// TIA Portal project "ANALOG INPUT" (V19)

(* hardware
DEVICE "SIMATIC 1200 station_1"  S71200.Device
   slot 0: "S7-1200 rack"  Rack  V1.0
   slot 1: "PLC_1"  CPU 1214C DC/DC/DC  6ES7 214-1AG40-0XB0  V4.0
   slot 3: "AQ1 x 12 bits_1"  6ES7 232-4HA30-0XB0  V1.0
DEVICE "HMI_1"  KTP600 Basic color PN
   slot 0: "HMI"  HMI  6AV6 647-0AD11-3AX0  12.0.0.0
   slot 1: "HMI_RT_1"  KTP600 Basic color PN  6AV6 647-0AD11-3AX0  12.0.0.0
   slot 5: "IE_CP_1"  PROFINET Interface  IE_CP  V7.1.0
      slot 1: "PROFINET_Interface_1"  PROFINET Interface
         slot 1: "PORT_1"  Port  1.0.0.0
*)

// ===== PLC "PLC_1"  CPU 1214C DC/DC/DC =====

DATA_BLOCK "Simulated Analog Input"   // DB1
{ S7_Optimized_Access := 'TRUE' }
VERSION : 0.1
   VAR
      HEIGHT_AI : Int;
   END_VAR
BEGIN
END_DATA_BLOCK

ORGANIZATION_BLOCK "Main"   // OB1, LAD, ProgramCycle
TITLE = "Main Program Sweep (Cycle)"
{ S7_Optimized_Access := 'TRUE' }
VERSION : 0.1
BEGIN
END_ORGANIZATION_BLOCK

(* ===== HMI "HMI_RT_1" =====
system functions are stored by id; their names below are inferred from use
connection "HMI_Connection_1": ETHERNET, SMART_S7_1200_OMS

HMI tags "Default tag table"
   "Conveyor_Control_DB_HEIGHT" : Int = PLC Conveyor_Control_DB.HEIGHT, 1 s
   "Simulated Analog Input_HEIGHT_AI" : Int = PLC "Simulated Analog Input".HEIGHT_AI, 1 s
   "ERROR" : Bool = PLC ERROR AT %Q0.1, 1 s
   "Conveyor_Control_DB_PART_A_ERROR" : Bool = PLC Conveyor_Control_DB.PART_A_ERROR, 1 s
   "Conveyor_Control_DB_PART_B_ERROR" : Bool = PLC Conveyor_Control_DB.PART_B_ERROR, 1 s

Template "Template_1" 320x240
   Softkey "Softkey_F6" at 266,202 size 53x38
      on KeyDown: StopRuntime(0)
   TextField "Template_Text field_1" at 280,208 size 34x27; Text 'F6 EXIT'

screen "Root screen" 320x240, template "Template_1"
   TextField "Text field_1" at 90,5 size 129x21; Text 'ANALOG INPUT'
   GraphicIOField "PlotLight_Square_R" at 38,62 size 25x25; PictureOff "PilotLight_Square_R_Off_256c"; PictureOn "PilotLight_Square_R_On_256c"
      ProcessValue <- "ERROR"
   TextField "Text field_2" at 209,43 size 78x16; Text 'Error Message'
   TextField "Text field_3" at 107,43 size 77x16; Text 'Gauge Height'
   TextField "Text field_4" at 26,40 size 45x16; Text 'ERROR'
   IOField "I/O field_1" at 110,65 size 71x22; FormatPattern 999
      ProcessValue <- "Conveyor_Control_DB_HEIGHT"
   TextField "Text field_5" at 211,65 size 75x16; Text 'Part A Error'
      Visibility <- "Conveyor_Control_DB_PART_A_ERROR"
   IOField "I/O field_2" at 124,154 size 70x36; FormatPattern 99999
      ProcessValue <- "Simulated Analog Input_HEIGHT_AI"
   Button "Button_1" at 235,174 size 36x36; TextOff 'Text'; PictureOff "Up_Arrow"
      on Press: function_dd21b452("Simulated Analog Input_HEIGHT_AI", 10)
   Button "Button_2" at 47,174 size 36x36; TextOff 'Text'; PictureOff "Down_Arrow"
      on Press: function_b9b71300("Simulated Analog Input_HEIGHT_AI", 10)
   Button "Button_3" at 274,154 size 36x36; TextOff 'Text'; PictureOff "Up_Arrow"
      on Press: function_dd21b452("Simulated Analog Input_HEIGHT_AI", 1000)
   Button "Button_4" at 196,154 size 36x36; TextOff 'Text'; PictureOff "Up_Arrow"
      on Press: function_dd21b452("Simulated Analog Input_HEIGHT_AI", 1)
   Button "Button_5" at 47,136 size 36x36; TextOff 'Text'; PictureOff "Down_Arrow"
      on Press: function_b9b71300("Simulated Analog Input_HEIGHT_AI", 100)
   Button "Button_6" at 86,154 size 36x36; TextOff 'Text'; PictureOff "Down_Arrow"
      on Press: function_b9b71300("Simulated Analog Input_HEIGHT_AI", 1)
   TextField "Text field_6" at 210,135 size 10x18; Text '1'
   TextField "Text field_7" at 244,207 size 18x18; Text '10'
   Button "Button_7" at 8,154 size 36x36; TextOff 'Text'; PictureOff "Down_Arrow"
      on Press: function_b9b71300("Simulated Analog Input_HEIGHT_AI", 1000)
   Button "Button_8" at 235,136 size 36x36; TextOff 'Text'; PictureOff "Up_Arrow"
      on Press: function_dd21b452("Simulated Analog Input_HEIGHT_AI", 100)
   TextField "Text field_8" at 239,119 size 26x18; Text '100'
   TextField "Text field_9" at 276,136 size 34x18; Text '1000'
   TextField "Text field_10" at 99,135 size 10x18; Text '1'
   TextField "Text field_11" at 56,207 size 18x18; Text '10'
   TextField "Text field_12" at 53,119 size 26x18; Text '100'
   TextField "Text field_13" at 8,136 size 34x18; Text '1000'
   TextField "Text field_14" at 114,123 size 93x28; Text 'ANALOG SENSOR BIT VALUE'
   TextField "Text field_15" at 99,196 size 126x15; Text 'Bit Range: 0 to 27648'
   TextField "Text field_16" at 211,65 size 74x16; Text 'Part B Error'
      Visibility <- "Conveyor_Control_DB_PART_B_ERROR"
*)